FUNCTION_BLOCK DIV_REAL (* IEC 61131-3 REAL Division *)
  (* Standard: 61131-3 *)
  (* Version 0.0, 2004-12-15, JHC, Rockwell Automation, Converted from SRC format. *)
  (* Compiler header: package fb.rt.plc.math; *)
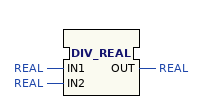
  VAR_INPUT
    IN1 : REAL; (* Dividend *)
    IN2 : REAL; (* Divisor *)
  END_VAR
  VAR_OUTPUT
    OUT : REAL; (* Quotient *)
  END_VAR
END_FUNCTION_BLOCK
